FUNCTION_BLOCK EL2032
VAR
	{attribute addProperty Name "WcState"}
	_wcState : WcStateInputToggle;
	{attribute addProperty Name "Info data"}
	_infoData : InfoDataBase;
	_io : EL2032_Data;
END_VAR

PROPERTY IO : REFERENCE TO EL2032_Data
GET
IO REF= _io;
END_GET
END_PROPERTY

PROPERTY WcState : REFERENCE TO WcStateInputToggle
GET
WcState REF= _wcState;
END_GET
END_PROPERTY

END_FUNCTION_BLOCK

(* stored: Version 1.1.0.1, ProductVersion 3.1.4024.9
   POU EL2032: Id {c9ac5850-9e39-0f29-39ae-8752722b4294}, SpecialFunc None
   Property IO: Id {f8913651-3560-06fd-1b13-eb5db7c0a545}
   Get Get: Id {c25f3e96-7b1e-01d7-12af-99479cfd2d18}
   Property WcState: Id {d0f3d198-7039-0356-0115-4457b7bac1bb}
   Get Get: Id {ed1ebc52-42e5-063f-121d-5d474b24b1e1} *)
